Staubli VAL3: cleanUpDataBase.pgx

program cleanUpDataBase()
  local num i
  local num j
  local num idx
  local string sAppList[50]
  local num nFoundIndex
  local string txt
begin
    //\brief
  //Remove database entries of non existing user applications.
  //
  // get the list of existing applications
  //\var i
  //\var j
  //\var idx
  //\var sAppList
  //\var nFoundIndex
  //\var txt
  //
//!brief
  //Remove database entries of non existing user applications.
  //
  // get the list of existing applications
  txt=""
  libList(txt,sRawList)
  idx=0
  for i=0 to size(sRawList)-1
    if find(sRawList[i],"a")==0
      sAppList[idx]=sRawList[i]
      idx=idx+1
    endIf
  endFor
  for j=0 to size(data:dbAppNameList)-1
    call list:indexOfString(sAppList,data:dbAppNameList[j],nFoundIndex)
    if nFoundIndex==-1 or data:dbAppNameList[j]=="" and j>0
      $ddel(data:dbPartCount,j)
      $ddel(data:dbPartReject,j)
      $ddel(data:dbAppDescList,j)
      $ddel(data:dbAppNameList,j)
    endIf
  endFor
end
